FUNCTION_BLOCK FB_PythonInterface EXTENDS T_NamedBase
VAR
  // interface paths (config)
  sPythonInterfacePath : STRING(255); //e.g. 'PRG_x.fb_PythonInterface'
  sPythonContainerPath : STRING(255); //e.g. 'PRG_x.fb_ContainerManager.sL_Containers[%id%].fb_ImageDeformation'
  sPythonScriptPath    : STRING(255);

	bPythonHeartbeat : BOOL;      // <- script is toggling this value as long as it's alive (for plc watchdog of script)
	nPythonPID : UDINT := 0;      // <- python process id (evaluated and given by external script)
  nPythonNewJob : DINT;         // -> new job indication to script
  bPythonNewJobDone : BOOL;     // <- new job registered/done by script

	nContainerToRegister : DINT := -1; // <- triggers a new container creation, except if < 0
  nContainerToRegister_mem : DINT := -1;
	nContainerToDelete : DINT := -1;   // <- triggers a new container deletion, except if < 0
  nContainerToDelete_mem : DINT := -1;
  
  //Job settings all in [px]
  nPythonImageOffsetY : UDINT := 0;     // [px]  y offset from 0 to source image
  nPythonImageWidth : UDINT := 1000;    // [px]  source image width (depth)
  nPythonImageHeight  : UDINT := 1000;  // [px]  source image height (width)
  //Grid settings
  nPythonGridPitchX  : UDINT := 100;    // [px]
  nPythonGridPitchY  : UDINT := 100;    // [px]
  nPythonGridSizeX   : UDINT := 0;      // (not yet used) number of grid columns
  nPythonGridSizeY   : UDINT := 0;      // (not yet used) number of grid rows
  //Cam specific settings
  nPythonCamFrameWidth  : UDINT := 200; // [px]
  
  nState : UDINT;
  fbStateTimer : TON;
  fBScriptLauncher : FB_ScriptLauncher;
  _bEnable : BOOL;
  _bKeepAlive : BOOL := TRUE; // keep script alive (restart after crash/close)
  _nStarts : UDINT;   // number of script start attempts
  _nErrCtr : UDINT;   // script error state counter
  _bBusy : BOOL;
  _nErrId : UDINT;
  _bJobStartRequest: BOOL;
  _bJobStopRequest: BOOL;
  _bResetError : BOOL;    // reset state machine error 
  _nJobIdCtr : DINT;
 
	// Python script heartbeat
	fbWatchdog : TOF;
	tWatchdogPeriod : TIME := T#1S;
	fbHeartbeat1 : R_TRIG;
	fbHeartbeat2 : F_TRIG;
	bScriptAlive : BOOL;

END_VAR

VAR CONSTANT
  cStateIdle      : UDINT := 0;
  cStateStartup   : UDINT := 10;
  cStartScript    : UDINT := 20;
  cStateRunning   : UDINT := 30;
  cStateJobActive : UDINT := 40;
  cStateError     : UDINT := 50;
  cStateStop      : UDINT := 60;
  cStateStopping  : UDINT := 70;
  
  cMaxStartAttempts : UDINT := 5;
END_VAR

InterfaceStateMachine();

// reset Container commands, so we suer have a change event on index
IF nContainerToRegister >= 0 AND nContainerToRegister_mem >= 0 THEN nContainerToRegister := -1; END_IF
IF nContainerToDelete >= 0 AND nContainerToDelete_mem >= 0 THEN nContainerToDelete := -1; END_IF
nContainerToRegister_mem := nContainerToRegister;
nContainerToDelete_mem := nContainerToDelete;

fbHeartbeat1(CLK := bPythonHeartbeat);
fbHeartbeat2(CLK := bPythonHeartbeat);
fbWatchdog(IN := fbHeartbeat1.Q OR fbHeartbeat2.Q, PT:=tWatchdogPeriod);
bScriptAlive := fbWatchdog.Q AND nPythonPID <> 0;

{attribute 'monitoring':='call'}
PROPERTY bBusy : BOOL
GET
bBusy := _bBusy;
END_GET
END_PROPERTY

PROPERTY bEnable : BOOL
GET
bEnable := _bEnable;
END_GET
SET
_bEnable := bEnable;
END_SET
END_PROPERTY

{attribute 'monitoring':='call'}
PROPERTY bError : BOOL
GET
IF nState = cStateError THEN bError := TRUE; END_IF;
END_GET
END_PROPERTY

{attribute 'monitoring':='call'}
PROPERTY bJobActive : BOOL
GET
IF nState = cStateJobActive THEN bJobActive := TRUE; END_IF;
END_GET
END_PROPERTY

{attribute 'monitoring':='call'}
PROPERTY bRunning : BOOL
GET
IF nState = cStateRunning THEN bRunning := TRUE; END_IF;
END_GET
END_PROPERTY

METHOD Init : BOOL
VAR_INPUT
  sCTManagerPath : T_MaxString;  // ct manager path (plc variable instance path)
  sScriptPath    : T_MaxString;  // path to python script base folder, e.g. C:\Work\script
END_VAR
sPythonInterfacePath := THIS^.InstanceName;
sPythonContainerPath := sCTManagerPath;
sPythonScriptPath    := sScriptPath;

// init launcher
fBScriptLauncher.Init(sPythonScriptPath);


//Launch init procedure
fbStateTimer(PT:=T#5S);
nState := cStateIdle;
END_METHOD

ACTION InterfaceStateMachine:

CASE(nState) OF
  // Idle
  cStateIdle  :
    _bJobStartRequest:=FALSE;
    _bJobStopRequest:=FALSE;
    IF bEnable THEN
      nState := cStateStartup;
    END_IF  

  //Startup
  cStateStartup   :
    fbStateTimer(IN:=TRUE);         // start timeout
    _bBusy := TRUE;

    IF fbStateTimer.Q THEN
      fbStateTimer(IN:=FALSE);
      _nStarts := _nStarts + 1;
      IF bScriptAlive THEN
        nState := cStateRunning;    // is already running
      ELSE  
        RunPythonScript();          // start script
        nState := cStartScript;
			END_IF
		END_IF
  
  //Start Python script and wait until it starts
  cStartScript    :
    fbStateTimer(IN:=TRUE);
    _bBusy := TRUE;

    IF NOT fBScriptLauncher.bBusy AND bScriptAlive THEN 
      IF fBScriptLauncher.bError THEN //Launch error
        LogError(F_Concat2('Script start error=', TO_STRING(fBScriptLauncher.nErrId)));
        nState := cStateError;
      ELSE //Launch done and heartbeat ok
        nState := cStateRunning;
        fbStateTimer(IN:=FALSE);
			END_IF
    ELSIF fbStateTimer.Q THEN //Timeout error
      LogError('Script start error');
      nState := cStateError;
		END_IF
 
  //Script running with correct watchdog feedback
  cStateRunning   : 
    fbStateTimer(IN:=_bJobStartRequest);
    _bBusy := _bJobStartRequest;
    _bJobStopRequest := FALSE;
    _nStarts := 0;
    
    IF _bJobStartRequest AND bPythonNewJobDone THEN
      _bJobStartRequest:=FALSE;
      bPythonNewJobDone := FALSE; 
      fbStateTimer(IN:=FALSE);  
      nState := cStateJobActive;
    ELSIF NOT bScriptAlive THEN //Watchdog error
      LogError('Script watchdog error');
      nState := cStateError;
    ELSIF fbStateTimer.Q THEN //Job timeout error
      LogError('Script new job done error');
      nState := cStateError;
    ELSIF NOT bEnable THEN
      nState := cStateStop;
		END_IF
  
  //JobStarted
  cStateJobActive :
    fbStateTimer(IN:=_bJobStopRequest);
    _bBusy := _bJobStopRequest;
    
    IF _bJobStopRequest THEN
      nPythonNewJob := 0;
    END_IF;  
    
    IF _bJobStopRequest THEN
      _bJobStopRequest:=FALSE;
      fbStateTimer(IN:=FALSE);  
      nState := cStateRunning;
    ELSIF NOT bScriptAlive THEN //Watchdog error
      LogError('Script watchdog error');
      nState := cStateError;
    ELSIF fbStateTimer.Q THEN //Job timeout error
      LogError('Script new job done error');
      nState := cStateError;
    ELSIF NOT bEnable THEN
      nState := cStateStop;
		END_IF
  
  //Error  
  cStateError     :
    fbStateTimer(IN:=FALSE);  
    _bJobStartRequest:=FALSE;
    _bJobStopRequest:=FALSE;
    IF _bResetError OR NOT bEnable OR (_bKeepAlive AND _nStarts <= cMaxStartAttempts)  THEN
      _bResetError := FALSE;
      _nErrCtr := _nErrCtr + 1;
      nState := cStateStop ;
		END_IF
    
  //Stop 
  cStateStop  :
    StopPythonScript();
    nState := cStateStopping;

  // Stopping
  cStateStopping  :
    IF NOT fBScriptLauncher.bBusy THEN 
      IF fBScriptLauncher.bError THEN //Launch error
        LogError(F_Concat2('Script stop errror:', TO_STRING(fBScriptLauncher.nErrId)));
			END_IF
      nState := cStateIdle;
    END_IF

END_CASE
END_ACTION

METHOD JobStart
VAR_INPUT
  nJobImageWidth : UDINT;
  nJobImageHeigth  : UDINT;
  nCamFrameWidth : UDINT;
  pGridSettings  : POINTER TO ST_DefGridSettings;
END_VAR
_bJobStartRequest := TRUE;
_nJobIdCtr := _nJobIdCtr + 1;
nPythonNewJob := _nJobIdCtr;


nPythonImageWidth := nJobImageWidth * GVL_Deformation.nC_GridSubReso;
nPythonImageHeight :=nJobImageHeigth * GVL_Deformation.nC_GridSubReso;
nPythonCamFrameWidth := nCamFrameWidth * GVL_Deformation.nC_GridSubReso;
IF pGridSettings <> 0 THEN
  nPythonImageOffsetY := pGridSettings^.nGridImageOffsetY * GVL_Deformation.nC_GridSubReso;
  nPythonGridPitchX := pGridSettings^.nGridPitchX * GVL_Deformation.nC_GridSubReso;
  nPythonGridPitchY := pGridSettings^.nGridPitchY * GVL_Deformation.nC_GridSubReso;
  nPythonGridSizeX := pGridSettings^.nGridSizeX * GVL_Deformation.nC_GridSubReso;
  nPythonGridSizeY := pGridSettings^.nGridSizeY * GVL_Deformation.nC_GridSubReso; 
END_IF
END_METHOD

METHOD JobStop : BOOL
VAR_INPUT
END_VAR
_bJobStopRequest:=TRUE;
END_METHOD

{attribute 'monitoring':='call'}
PROPERTY nErrorId : UDINT
GET
nErrorId := _nErrId;
END_GET
END_PROPERTY

(*
  Register CT to script.
  :return: TRUE if success.
*)
METHOD RegisterCT : BOOL
VAR_INPUT
  nCTIdx  : UDINT;  // ct memory index
END_VAR
IF NOT bScriptAlive THEN RETURN; END_IF  // script not ready, ignore request

nContainerToRegister := UDINT_TO_DINT(nCTIdx);
RegisterCT := TRUE;
END_METHOD

METHOD RemoveCT : BOOL
VAR_INPUT
    nCTID : UDINT;
END_VAR
IF NOT bScriptAlive THEN RETURN; END_IF  // script not ready, ignore request

nContainerToDelete := UDINT_TO_DINT(nCTID);

RemoveCT := TRUE;
END_METHOD

METHOD PRIVATE RunPythonScript : BOOL
VAR_INPUT
END_VAR
VAR
  ams_host : STRING;
  ams_port : UINT;
  cmd : STRING;
END_VAR
// config launcher cmd line for script
//   e.g. fBScriptLauncher.Start('172.17.7.143.1.1 851 PRG_PRINT.fbWorkerDefGrid_Python.fbPythonInterface --sim_mode');

// get parameter dynamically
ams_host := PRG_SYSTEMBASE.sO_AmsNetIdLocalHost;  // localhost
ams_port := TwinCAT_SystemInfoVarList._AppInfo.AdsPort;
cmd := F_Concat5(ams_host,' ',TO_STRING(ams_port),' ',sPythonInterfacePath);
fBScriptLauncher.sStartScriptName := 'start.bat';
fBScriptLauncher.sStopScriptName  := 'stop.bat';
fBScriptLauncher.Start(cmd);
END_METHOD

METHOD PRIVATE StopPythonScript
VAR_INPUT
END_VAR
fBScriptLauncher.Stop(nPID := THIS^.nPythonPID);
END_METHOD

{attribute 'monitoring':='call'}
PROPERTY tWatchdogTime : TIME
GET
tWatchdogTime := fbWatchdog.ET;
END_GET
END_PROPERTY

END_FUNCTION_BLOCK

(* stored: Version 1.1.0.1, ProductVersion 3.1.4024.3
   POU FB_PythonInterface: Id {32bc7ee3-797a-48a1-b6c9-938bdbb76439}, SpecialFunc None
   Property bBusy: Id {15ecb802-f104-48b3-a8e9-296585ddbd3b}
   Get Get: Id {139a7e3b-71b0-4b41-a84c-6f1ce8c1465e}
   Property bEnable: Id {a328260d-f3bb-44ce-926f-19d84ae50bc4}
   Get Get: Id {c3e54d05-49b9-49b2-afe1-2edeba063599}
   Set Set: Id {a5cb12de-b348-4aa0-ac98-f1624d50cea7}
   Property bError: Id {6f1a5717-89e4-48eb-b728-b4de0dccc9aa}
   Get Get: Id {22606d90-35e2-46d9-b94a-3ab7829f7825}
   Property bJobActive: Id {19e50aac-19c8-4473-8fa4-8f452084848d}
   Get Get: Id {ca400b3a-23f2-429e-82ed-973227f5ccba}
   Property bRunning: Id {e1d4af5a-cce0-4b67-86b9-9f5d618aeda0}
   Get Get: Id {3f2c9f1a-dad5-4a1b-b301-6b9ceb3c89c2}
   Method Init: Id {5691349d-c567-4cf4-a8d6-db318033dadf}
   Action InterfaceStateMachine: Id {235b0a93-bff5-4257-b33a-44f1b952b745}
   Method JobStart: Id {8405a1de-7ba0-408e-bd94-f023aa4d1d8c}
   Method JobStop: Id {a622984e-d634-417d-9233-aba88648edec}
   Property nErrorId: Id {45601785-2b9c-481d-be8c-9623ba129752}
   Get Get: Id {4e03f40b-d6e1-4626-8168-625f45ef2c79}
   Method RegisterCT: Id {d26fde14-0d98-487d-b756-8dec552ded5f}
   Method RemoveCT: Id {28d59eb6-90bf-4722-adc3-86b27e084ab5}
   Method RunPythonScript: Id {eef5e660-c4a2-454d-95d6-7e90dbff3075}
   Method StopPythonScript: Id {c21082da-2f62-4d93-8645-06b9e715913a}
   Property tWatchdogTime: Id {27534f97-fbe5-46f4-9a92-902b4b859dbf}
   Get Get: Id {e7f80b61-e2e0-44d3-8b4e-f911a33f84d0} *)
